FUNCTION_BLOCK Q_NumericValue_PHYSA (* Command change numeric value — accepts physical REAL value via AR adapter (wraps Q_NumericValue_PHYS) *)
  (* Standard: ISO 11783-6; Description: Copyright (c) 2026 Meisterschulen am Ostbahnhof This program and the accompanying materials are made available under the terms of the Eclipse Public License 2.0 which is available at https://www.eclipse.org/legal/epl-2.0/ SPDX-License-Identifier: EPL-2.0 *)
  (* Version 1.0, 2026-04-14, Franz Höpfinger, Meisterschulen am Ostbahnhof *)
  PACKAGE isobus::UT::Q;
  IMPORT eclipse4diac::core::TypeHash;
  IMPORT logiBUS::utils::conversion::phys::NumericObjectPool_S;
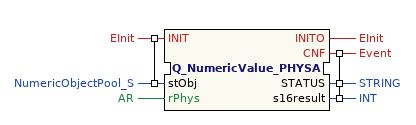
  EVENT_INPUT
    INIT : EInit WITH stObj; (* Service Initialization *)
  END_EVENT
  EVENT_OUTPUT
    INITO : EInit; (* Initialization Confirm *)
    CNF WITH STATUS, s16result; (* Confirmation of Requested Service *)
  END_EVENT
  VAR_INPUT
    stObj : logiBUS::utils::conversion::phys::NumericObjectPool_S; (* Object pool properties (u16ObjId, scale, offset, decimals) *)
  END_VAR
  VAR_OUTPUT
    STATUS : STRING; (* Service Status *)
    s16result : INT; (* retval see Q_NumericValue *)
  END_VAR
  SOCKETS
    rPhys : adapter::types::unidirectional::AR; (* Physical REAL value input *)
  END_SOCKETS
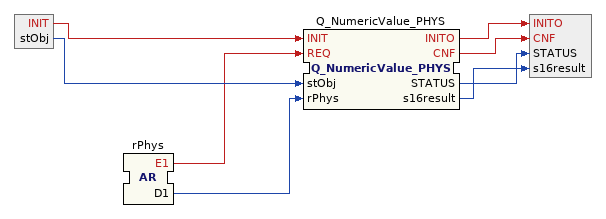
  FBS
    Q_NumericValue_PHYS : isobus::UT::Q::Q_NumericValue_PHYS;
  END_FBS
  EVENT_CONNECTIONS
    INIT TO Q_NumericValue_PHYS.INIT;
    rPhys.E1 TO Q_NumericValue_PHYS.REQ;
    Q_NumericValue_PHYS.INITO TO INITO;
    Q_NumericValue_PHYS.CNF TO CNF;
  END_CONNECTIONS
  DATA_CONNECTIONS
    stObj TO Q_NumericValue_PHYS.stObj;
    rPhys.D1 TO Q_NumericValue_PHYS.rPhys;
    Q_NumericValue_PHYS.STATUS TO STATUS;
    Q_NumericValue_PHYS.s16result TO s16result;
  END_CONNECTIONS
END_FUNCTION_BLOCK
